{attribute 'GeneratedUsingTerminal: EL3612-0000-0016'}
{attribute addProperty BoxType "EL3612-0000-0016"}
{attribute addProperty Id "EtcSlaveTerminalBaseAI_Inputs_Channel_1AT %I*AI_Inputs_Channel_10B8F80A11AI_Inputs_Channel_2AT %I*AI_Inputs_Channel_10B8F80A11WcStateAT %I*WcState_9091E0EB2InfoDataAT %I*InfoData_32EB74EA10"}
{attribute addProperty CRC "810058752"}
{attribute addProperty Size "34"}
TYPE EL3612_30488400 EXTENDS EtcSlaveTerminalBase :
STRUCT
	{attribute addProperty Name "AI_Inputs_Channel_1"}
	AI_Inputs_Channel_1 : AI_Inputs_Channel_10B8F80A;
	{attribute addProperty Name "AI_Inputs_Channel_2"}
	AI_Inputs_Channel_2 : AI_Inputs_Channel_10B8F80A;
	{attribute addProperty Name "WcState"}
	WcState : WcState_9091E0EB;
	{attribute addProperty Name "InfoData"}
	InfoData : InfoData_32EB74EA;
END_STRUCT
END_TYPE

(* stored: Version 1.2.0.0, ProductVersion 3.1.4024.9
   DUT EL3612_30488400: Id {bbc25898-8234-4b5b-993f-1614913c5cbf} *)
